PROGRAM MAIN
VAR
	State			  : USINT;
	LocalLogger		  : SimpleLocalLogger;
	Message			  : SimpleLogMessage;
	Source			  : SimpleLogSource;
	LogAMessage		  : BOOL;
	IndividualMessage : BOOL;
END_VAR

CASE State OF
	0:
		GVL.Logger.Subscribe(LocalLogger);
		State := 10;

	10:
END_CASE

IF LogAMessage THEN
	LogAMessage := FALSE;
	GVL.Logger.LogMessage(Source, Message);
END_IF

IF IndividualMessage THEN
	IndividualMessage := FALSE;
	GVL.Logger.LogMessageIndividual(Message := 'My Individual Message');
END_IF

END_PROGRAM

(* stored: Version 1.1.0.1
   POU MAIN: Id {ca8aab67-3a8c-46ae-a624-30d4645d11d7}, SpecialFunc None *)
